FUNCTION_BLOCK ObjectTestSuite
VAR
	ReRun : BOOL;
	ObjTestSuite : TestSuite<TestSuiteParameter.MaxTestCount>('C:\ProgramData\Beckhoff\TwinCAT\3.1\Boot\Object_Tests.xml') := (TestSuiteName := 'Object Test Suite');
END_VAR

ObjectAcceptsName_Test();
IF ReRun THEN
	ObjTestSuite.ReRunTests();
	ReRun := FALSE;
END_IF

METHOD ObjectAcceptsName_Test
VAR_INST
	Expected : BOOL := TRUE;
	Actual	 : BOOL;
END_VAR
VAR
	TestMockObj : MockObject(Name := 'Bob');
END_VAR
IF ObjTestSuite.Test(__POUNAME()).ExecuteTest() THEN
	Expected := TRUE;
	Actual := TestMockObj.Name = 'Bob';
	ObjTestSuite.Test(__POUNAME()).AssertEqual(Expected, Actual);
END_IF
END_METHOD

END_FUNCTION_BLOCK

(* stored: Version 1.1.0.1
   POU ObjectTestSuite: Id {dff4e0f5-e147-4a10-a1c9-bb53cdb042da}, SpecialFunc None
   Method ObjectAcceptsName_Test: Id {41bba9a9-9474-43ec-888e-ea41aff17b51} *)
